FUNCTION_BLOCK T_CommandQueue_GetNextCommanHighPriorityWithNormalPriority_ReturnTrue EXTENDS T_UnitTestBase
VAR
  commandHighPriority : T_CommandTask;
  commandNormalPriority : T_CommandTask;
  commandQueue : T_CommandQueue;
  myTestState, prevState : (ARRANGE, ACT, ASSERT);
  actual : I_Task;
  expected : I_Task;
END_VAR

CASE myTestState OF
  ARRANGE:
  	expected := commandHighPriority;
	commandQueue.Clear();
	commandQueue.AddNormalPriority(commandNormalPriority);
	commandQueue.AddHighPriority(commandHighPriority);
    myTestState := ACT;
  
  ACT:
    commandQueue.GetNext(output_command => actual);
	myTestState := ASSERT;
	
  ASSERT:
    assertion.AssertEquals_INTERFACE(expected, actual, 'commandQueue.GetNext high priority with Low priority = TRUE');
    myTestState := ARRANGE;
    TestFinished();
END_CASE

END_FUNCTION_BLOCK

(* stored: Version 1.1.0.1, ProductVersion 3.1.4024.12
   POU T_CommandQueue_GetNextCommanHighPriorityWithNormalPriority_ReturnTrue: Id {5a88bb6b-1526-492f-afaf-f386ba6c0e3a}, SpecialFunc None *)
